TYPE ST_VGC :
STRUCT

(* Readbacks *)
	i_xOpnLS	: BOOL;
	i_xClsLS	: BOOL;

(* EPICS Controls *)
	xOPN_SW	: BOOL;
	xAlmRst	: BOOL;
	xOvrdOpn	:	BOOL;

(* Interlocks *)
	xDP_OK	:	BOOL;	(* Managed by the VGC function (FB_VGC) *)
	xEXT_OK	:	BOOL := FALSE;	(* External interlock for custom interlocking in addition to regular DP ilk, this must be set true, or the interlock condition before calling the FB_VGC *)
	xOPN_OK	:	BOOL;	(* Final SUM of DP_OK and EXT_OK, needed because it allows the DP ilk to be switched off, see FB_VGC.Dis_DPIlk *)

(* Controls *)
	xOPN_DO	: BOOL;

(* Alarm Outpus *)
	xERR_DifPres		: 	BOOL;
	xERR_LstVac		: 	BOOL;
	xAlmSum			: 	BOOL;

END_STRUCT
END_TYPE

(* stored: Version 1.1.0.1, ProductVersion 3.1.4018.5
   DUT ST_VGC: Id {2c4a7ba8-0fa6-4a25-9ffd-90841b7d250a} *)
